KUKA KRL data list: vw_config.dat

&ACCESS RV
&PARAM TPVW_VERSION=8.3.17
DEFDAT VW_CONFIG PUBLIC

;FOLD USER GLOBALS;%E{E},%P___$$$___CONFIG.USB___start___
;==================================
; Userdefined Types
;==================================
;==================================
; Userdefined Externals
;==================================
;==================================
; Userdefined Variables
;==================================
;ENDFOLD;___$$$___CONFIG.USB___end_____

ENDDAT
